# EPICS autosave request: DG645/iocBoot/iocDG645-IOC-01/auto_settings.req
file "configMenu_settings.req" "P=$(P)AS:$(R),CONFIG=dgconfig"
file "drvDG645_settings.req" "P=$(P),R=$(R)"
